TYPE ST_HEATER_HMI :
STRUCT
	state:			ST_HEATER_STATE;
	service:		ST_HEATER_SERVICE;
	settings:		ST_HEATER_SETTINGS;
	
	ai:				ST_AI_HMI;
	thermostat:		ST_THERMOSTAT_HMI;
END_STRUCT
END_TYPE

(* stored: Version 1.1.0.1
   DUT ST_HEATER_HMI: Id {00de9a9e-29a6-4e5d-aca1-c7c0afb19a90} *)
